(* This Function block is for the BALLUF sensor *)
FUNCTION_BLOCK FB_Balluff_BMF00LA
VAR
	In		AT %I* 	: ST_Balluff_BMF00LA_Status;
END_VAR

END_FUNCTION_BLOCK

(* stored: Version 1.1.0.1, ProductVersion 3.1.4024.12
   POU FB_Balluff_BMF00LA: Id {ec4aac2a-536b-48d3-8449-df4ef6428802}, SpecialFunc None *)
